SUBAPPLICATION Uebung_020d (* DigitalInput_I1 auf DigitalOutput_Q1; TOF Ausschaltverzögert; aufgelöst *)
  (* Standard: 61499-2; Description: Copyright (c) 2023 Meisterschulen am Ostbahnhof This program and the accompanying materials are made available under the terms of the Eclipse Public License 2.0 which is available at https://www.eclipse.org/legal/epl-2.0/ SPDX-License-Identifier: EPL-2.0 *)
  (* Version 1.0, 2023-10-23, Franz Höpfinger, Meisterschulen am Ostbahnhof, initial API and implementation and/or initial documentation *)
  PACKAGE Uebungen;
  IMPORT logiBUS::io::DI::logiBUS_DI::Input_I1;
  IMPORT logiBUS::io::DQ::logiBUS_DO::Output_Q1;
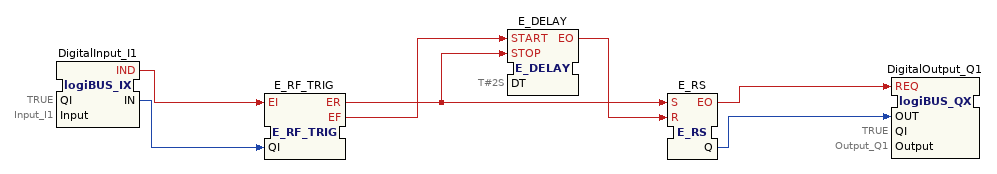
  FBS
    DigitalOutput_Q1 : logiBUS::io::DQ::logiBUS_QX(QI := TRUE, Output := Output_Q1);
    DigitalInput_I1 : logiBUS::io::DI::logiBUS_IX(QI := TRUE, Input := Input_I1);
    E_RF_TRIG : iec61499::events::E_RF_TRIG;
    E_RS : iec61499::events::E_RS;
    E_DELAY : iec61499::events::E_DELAY(DT := T#2S);
  END_FBS
  EVENT_CONNECTIONS
    DigitalInput_I1.IND TO E_RF_TRIG.EI;
    E_RS.EO TO DigitalOutput_Q1.REQ;
    E_RF_TRIG.ER TO E_RS.S;
    E_RF_TRIG.EF TO E_DELAY.START;
    E_DELAY.EO TO E_RS.R;
    E_RF_TRIG.ER TO E_DELAY.STOP;
  END_CONNECTIONS
  DATA_CONNECTIONS
    DigitalInput_I1.IN TO E_RF_TRIG.QI;
    E_RS.Q TO DigitalOutput_Q1.OUT;
  END_CONNECTIONS
END_SUBAPPLICATION
